// TIA Portal project "Linear Data Types" (V16)

(* hardware
DEVICE "S7-1200 station_1"  S7-1200 Station
   slot 0: "Rack_0"  S7-1200 Rack  Rack  V1.0
   slot 1: "PLC_1"  CPU 1212C DC/DC/DC  6ES7 212-1AE40-0XB0  V4.4
*)

// ===== PLC "PLC_1"  CPU 1212C DC/DC/DC =====

VAR_GLOBAL   // PLC tag table "Default tag table"
   "System_Byte" AT %MB1 : Byte;
   "FirstScan" AT %M1.0 : Bool;
   "DiagStatusUpdate" AT %M1.1 : Bool;
   "AlwaysTRUE" AT %M1.2 : Bool;
   "AlwaysFALSE" AT %M1.3 : Bool;
   "Clock_Byte" AT %MB0 : Byte;
   "Clock_10Hz" AT %M0.0 : Bool;
   "Clock_5Hz" AT %M0.1 : Bool;
   "Clock_2.5Hz" AT %M0.2 : Bool;
   "Clock_2Hz" AT %M0.3 : Bool;
   "Clock_1.25Hz" AT %M0.4 : Bool;
   "Clock_1Hz" AT %M0.5 : Bool;
   "Clock_0.625Hz" AT %M0.6 : Bool;
   "Clock_0.5Hz" AT %M0.7 : Bool;
END_VAR

TYPE "Int.ArrayPlus.UDT"
   STRUCT
      length : DInt;
      data : Array[0..4] of Int;
   END_STRUCT;
END_TYPE

DATA_BLOCK "Debug"   // DB1
{ S7_Optimized_Access := 'TRUE' }
VERSION : 0.1
   VAR
      pop_request : Bool;
      pop_value : Int;
      push_request : Bool;
      push_value : Int;
      push_message : String;
      shift_right_request : Bool;
      shift_right_places : DInt;
      shift_left_request : Bool;
      shift_left_places : DInt;
   END_VAR
BEGIN
END_DATA_BLOCK

DATA_BLOCK "Buffer"   // DB2
{ S7_Optimized_Access := 'TRUE' }
VERSION : 0.1
BEGIN
END_DATA_BLOCK

FUNCTION "Initializer" : Void   // FC1, SCL
{ S7_Optimized_Access := 'TRUE' }
VERSION : 0.1
   VAR_TEMP
      i : DInt;
   END_VAR
BEGIN
   (*
   FOR #i := 0 TO UDINT_TO_DINT("Int.Array.CountOfElement"("Buffer".data)) - 1 DO
       "Buffer".data[#i] := DINT_TO_INT(#i) + 1;
   END_FOR;

   "Debug".push_value := 1;
   *)

   FOR #i := 0 TO UDINT_TO_DINT("Int.Array.CountOfElement"("Buffer".data)) - 1 DO
       "Debug".push_message := "Int.ArrayPlus.Push"(value := 23 * DINT_TO_INT(#i + 1), buffer := "Buffer");
   END_FOR;
END_FUNCTION

FUNCTION "Int.ArrayPlus.Push" : String   // FC2, SCL
{ S7_Optimized_Access := 'TRUE' }
VERSION : 0.1
   VAR_INPUT
      value : Int;
   END_VAR
   VAR_IN_OUT
      buffer : "Int.ArrayPlus.UDT";
   END_VAR
   VAR_TEMP
      size : DInt;
   END_VAR
   VAR CONSTANT
      FULL : String := 'array full, no push';
      SUCCESS : String := 'success';
   END_VAR
BEGIN
   REGION "NO PUSH"
       #size := UDINT_TO_DINT("Int.Array.CountOfElement"(#buffer.data));
       IF #buffer.length = #size THEN
           #"Int.ArrayPlus.Push" := #FULL;
           RETURN;
       END_IF;
   END_REGION


   REGION "PUSH"
       // shift
       "Int.Array.ShiftRight"(places := 1,
                              data := #buffer.data);
       // save to leftmost
       #buffer.data[0] := #value;
       // increment length
       #buffer.length += 1;
       // return message
       #"Int.ArrayPlus.Push" := #SUCCESS;
       RETURN;
   END_REGION
END_FUNCTION

FUNCTION "Int.Array.ShiftRight" : Void   // FC3, SCL
{ S7_Optimized_Access := 'TRUE' }
VERSION : 0.1
   VAR_INPUT
      places : DInt;   // must be positive
   END_VAR
   VAR_IN_OUT
      data : Array[*] of Int;
   END_VAR
   VAR_TEMP
      i : DInt;
      size : DInt;
   END_VAR
BEGIN
   REGION "PRE CONDITION"
       IF #places <= 0 THEN
           RETURN;
       END_IF;
   END_REGION


   REGION "GET SIZE"    
       #size := UDINT_TO_DINT("Int.Array.CountOfElement"(#data));
   END_REGION


   REGION "FILL CONDITION"
       IF #places >= #size THEN
           "Int.Array.Fill"(value := 0,
                            data := #data);
           RETURN;
       END_IF;

   END_REGION


   REGION "SHIFT"
       FOR #i := #size - 1 TO 0 BY -1 DO
           // pre conditions
           IF #i < 0 THEN
               EXIT;
           END_IF;
           IF #i - #places < 0 THEN
               EXIT;
           END_IF;
           // shift
           #data[#i] := #data[#i - #places];
       END_FOR;
   END_REGION


   REGION "CORRECT DUPLICATION"
       FOR #i := 0 TO #places - 1 DO
           #data[#i] := 0;
       END_FOR;
   END_REGION


   REGION "RETURN"
   END_REGION
END_FUNCTION

FUNCTION "Int.Array.Fill" : Void   // FC4, SCL
{ S7_Optimized_Access := 'TRUE' }
VERSION : 0.1
   VAR_INPUT
      value : Int;   // value that will fill array
   END_VAR
   VAR_IN_OUT
      data : Array[*] of Int;
   END_VAR
   VAR_TEMP
      i : DInt;
      size : DInt;
   END_VAR
BEGIN
   #size := UDINT_TO_DINT("Int.Array.CountOfElement"(#data));
   FOR #i := 0 TO #size - 1 DO
       #data[#i] := #value;
   END_FOR;
   RETURN;
END_FUNCTION

FUNCTION "Int.Array.CountOfElement" : UDInt   // FC5, SCL
{ S7_Optimized_Access := 'TRUE' }
VERSION : 0.1
   VAR_INPUT
      data : Variant;
   END_VAR
BEGIN
   #"Int.Array.CountOfElement" := CountOfElements(#data);
   RETURN;
END_FUNCTION

FUNCTION "Int.ArrayPlus.Pop" : Int   // FC6, SCL
{ S7_Optimized_Access := 'TRUE' }
VERSION : 0.1
   VAR_IN_OUT
      buffer : "Int.ArrayPlus.UDT";
   END_VAR
   VAR_TEMP
      value : Int;
   END_VAR
BEGIN
   REGION "EMPTY"
       IF #buffer.length = 0 THEN
           #"Int.ArrayPlus.Pop" := 0;
           RETURN;
       END_IF;
   END_REGION


   REGION "NOT EMPTY"
       // save value
       #value := #buffer.data[0];
       // shift left
       "Int.Array.ShiftLeft"(places := 1,
                             data := #buffer.data);
       // decrement length
       #buffer.length -= 1;
       // return value
       #"Int.ArrayPlus.Pop" := #value;
       RETURN;
   END_REGION
END_FUNCTION

FUNCTION "Int.Array.ShiftLeft" : Void   // FC7, SCL
{ S7_Optimized_Access := 'TRUE' }
VERSION : 0.1
   VAR_INPUT
      places : DInt;   // must be positive
   END_VAR
   VAR_IN_OUT
      data : Array[*] of Int;
   END_VAR
   VAR_TEMP
      i : DInt;
      size : DInt;
   END_VAR
BEGIN
   REGION "PRE CONDITION"
       IF #places <= 0 THEN
           RETURN;
       END_IF;
   END_REGION


   REGION "GET SIZE"    
       #size := UDINT_TO_DINT("Int.Array.CountOfElement"(#data));
   END_REGION


   REGION "FILL CONDITION"
       IF #places >= #size THEN
           "Int.Array.Fill"(value := 0,
                            data := #data);
           RETURN;
       END_IF;

   END_REGION


   REGION "SHIFT"
       FOR #i := 0 TO #size - 1 DO
           // pre condition
           IF #i + #places > #size - 1 THEN
               EXIT;
           END_IF;
           // shift
           #data[#i] := #data[#i + #places];
       END_FOR;
   END_REGION


   REGION "CORRECT DUPLICATION"
   FOR #i := (#size - 1) TO (#size - #places) DO
           #data[#i] := 0;
       END_FOR;
   END_REGION


   REGION "RETURN"
       RETURN;
   END_REGION
END_FUNCTION

ORGANIZATION_BLOCK "Main"   // OB1, LAD, ProgramCycle
TITLE = "Main Program Sweep (Cycle)"
{ S7_Optimized_Access := 'TRUE' }
VERSION : 0.1
   VAR_INPUT
      Initial_Call : Bool;   // Initial call of this OB
      Remanence : Bool;   // =True, if remanent data are available
   END_VAR
   VAR_TEMP   // added for the SCL form of the ladder/FBD networks
      _w1 : Bool;
   END_VAR
BEGIN

REGION Network 1: INITIALIZE
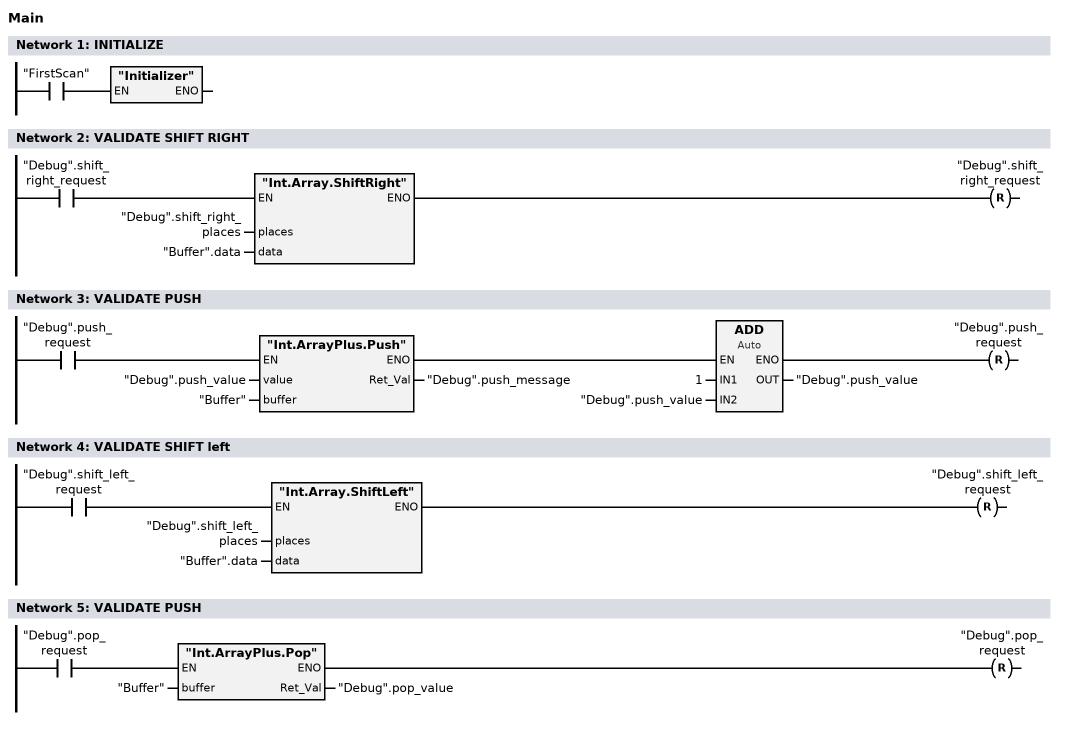
   RUNG wire#powerrail
      Contact( "FirstScan" )
      "Initializer"()
   END_RUNG
   // the same network as SCL:
   IF "FirstScan" THEN "Initializer"(); END_IF;
END_REGION

REGION Network 2: VALIDATE SHIFT RIGHT
   RUNG wire#powerrail
      Contact( "Debug".shift_right_request )
      "Int.Array.ShiftRight"(places := "Debug".shift_right_places, data := "Buffer".data)
      R_Coil( "Debug".shift_right_request )
   END_RUNG
   // the same network as SCL:
   "Int.Array.ShiftRight"(EN := "Debug".shift_right_request,
                          places := "Debug".shift_right_places,
                          data := "Buffer".data,
                          ENO => #_w1);
   IF #_w1 THEN "Debug".shift_right_request := FALSE; END_IF;
END_REGION

REGION Network 3: VALIDATE PUSH
   RUNG wire#powerrail
      Contact( "Debug".push_request )
      "Int.ArrayPlus.Push"(value := "Debug".push_value, buffer := "Buffer", Ret_Val => "Debug".push_message)
      Add(in1 := 1, in2 := "Debug".push_value, out => "Debug".push_value)
      R_Coil( "Debug".push_request )
   END_RUNG
   // the same network as SCL:
   "Debug".push_message := "Int.ArrayPlus.Push"(EN := "Debug".push_request,
                           value := "Debug".push_value,
                           buffer := "Buffer",
                           ENO => #_w1);
   IF #_w1 THEN
       "Debug".push_value := 1 + "Debug".push_value;
       "Debug".push_request := FALSE;
   END_IF;
END_REGION

REGION Network 4: VALIDATE SHIFT left
   RUNG wire#powerrail
      Contact( "Debug".shift_left_request )
      "Int.Array.ShiftLeft"(places := "Debug".shift_left_places, data := "Buffer".data)
      R_Coil( "Debug".shift_left_request )
   END_RUNG
   // the same network as SCL:
   "Int.Array.ShiftLeft"(EN := "Debug".shift_left_request,
                         places := "Debug".shift_left_places,
                         data := "Buffer".data,
                         ENO => #_w1);
   IF #_w1 THEN "Debug".shift_left_request := FALSE; END_IF;
END_REGION

REGION Network 5: VALIDATE PUSH
   RUNG wire#powerrail
      Contact( "Debug".pop_request )
      "Int.ArrayPlus.Pop"(buffer := "Buffer", Ret_Val => "Debug".pop_value)
      R_Coil( "Debug".pop_request )
   END_RUNG
   // the same network as SCL:
   "Debug".pop_value := "Int.ArrayPlus.Pop"(EN := "Debug".pop_request, buffer := "Buffer", ENO => #_w1);
   IF #_w1 THEN "Debug".pop_request := FALSE; END_IF;
END_REGION
END_ORGANIZATION_BLOCK